ABB RAPID module: Wobj_wobj_B2.mod

MODULE Wobj_wobj_B2
	! Points are read in order of declaration.
  ! Please do not change the order of points!

  LOCAL PERS robtarget pWobj_U_PointX1:=[[-106.496,-1451.867,-663.3867],[0.00554098561406136,-0.690757751464844,-0.723015487194061,-0.00846425537019968],[-2,0,-1,0],[0,9E+09,9E+09,9E+09,9E+09,9E+09]];
	LOCAL PERS robtarget pWobj_U_PointX2:=[[-71.90632,-2255.883,-665.711],[0.00554164405912161,-0.690758764743805,-0.7230144739151,-0.00846508145332336],[-2,0,-1,0],[0,9E+09,9E+09,9E+09,9E+09,9E+09]];
	LOCAL PERS robtarget pWobj_U_PointY1:=[[529.7682,-2228.682,-660.6664],[0.00553571060299873,-0.690758883953094,-0.7230144739151,-0.00846320576965809],[-1,0,0,0],[0,9E+09,9E+09,9E+09,9E+09,9E+09]];

ENDMODULE
